// TIA Portal V19 export
TYPE "FeedMachine_Config"
// stored: Access Published
   STRUCT
      SLS_VEL : LReal := 6000.0;
      DelayMissingCondition { ExternalVisible := 'False'} : Time := T#3s;   // Delay before rise up missing condition warnings
      Ax : Struct
         LeadScrewPitchVal : LReal := 1.0;
         MotorRevolution : LReal := 1.0;
         LoadRevolution : LReal := 1.0;
         PowerOffDelay : Time;
         StandstillVelocity : Real;
         StandstillDelay : Time;
      END_STRUCT;
      Fan : Struct
         Exist : Bool := FALSE;
         DelayOff : Time := T#10M;
      END_STRUCT;
      Brake_Presence : Bool;
   END_STRUCT;
END_TYPE
